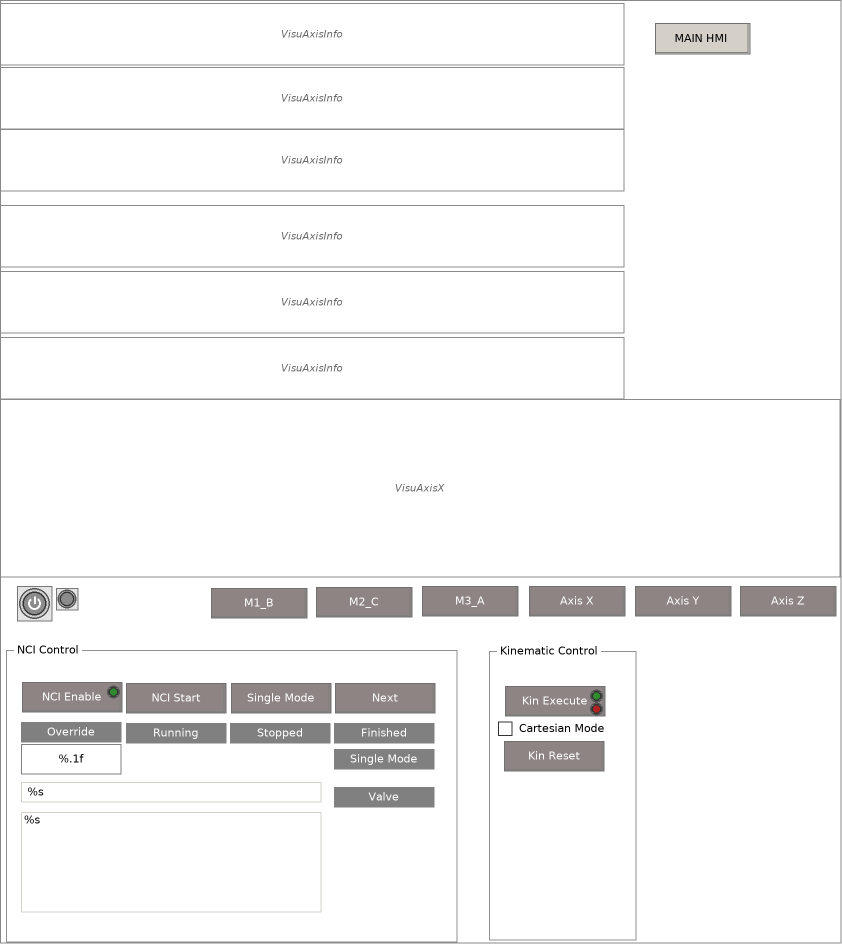
VISUALIZATION Visualization  // 842x944
    Frame (0,205 624x62)
        shows VisuAxisInfo(sAxisName := sAxisXName, stAxisRefVisu := AxisX)
    Frame (0,271 624x62)
        shows VisuAxisInfo(sAxisName := sAxisYName, stAxisRefVisu := AxisY)
    Frame (0,337 624x62)
        shows VisuAxisInfo(sAxisName := sAxisZName, stAxisRefVisu := AxisZ)
    Frame (0,399 840x178)
        shows VisuAxisX()
        shows VisuAxisY()
        shows VisuAxisZ()
        shows VisuAxisM1()
        shows VisuAxisM2()
        shows VisuAxisM3()
    Button (529,586 96x30), "Axis X"
        OnMouseClick: FrameSelectionChange Selection=SelectedFrame=c36eaae5-f889-4027-b551-56d3c927f334, GlobSel=AssignType=Directly, SelType=Locally
    Button (635,586 96x30), "Axis Y"
        OnMouseClick: FrameSelectionChange Selection=SelectedFrame=c36eaae5-f889-4027-b551-56d3c927f334, Selection=1, GlobSel=AssignType=Directly, SelType=Locally
    Button (740,586 96x30), "Axis Z"
        OnMouseClick: FrameSelectionChange Selection=SelectedFrame=c36eaae5-f889-4027-b551-56d3c927f334, Selection=2, GlobSel=AssignType=Directly, SelType=Locally
    GroupBox (6,642 451x300), "NCI Control"
        Button (16,40 100x30), "NCI Enable"
            toggle PRG_NcControl.bNciEnable
        Textfield (15,170 300x100), "%s", text variable: PRG_NcControl.sNciLines
        Button (225,41 100x30), "Single Mode"
            toggle PRG_NcControl.bNciSingleMode
        Rectangle (15,102 100x30), "%.1f", text variable: PRG_NcControl.fNciOverride
            OnMouseClick: write the text variable via VisuDialogs.Numpad
        Rectangle (15,80 100x20), "Override"
        Rectangle (120,81 100x20), "Running", colour toggle: PRG_NcControl.bProgramRunning
        Rectangle (224,81 100x20), "Stopped", colour toggle: PRG_NcControl.bProgramStopped
        Rectangle (328,81 100x20), "Finished", colour toggle: PRG_NcControl.bProgramFinished
        Rectangle (328,145 100x20), "Valve", colour toggle: PRG_MFuncControl.bTestValveOutput
        Button (120,41 100x30), "NCI Start"
            toggle PRG_NcControl.bNciStart
        Button (329,41 100x30), "Next"
            tap PRG_NcControl.bNciNextStep
        Rectangle (328,107 100x20), "Single Mode", colour toggle: PRG_NcControl.bSingleModeActive
        Lamp1 (100,42 15x16), variable: PRG_NcControl.bBuildGroupDone, style: Lamp-Lamp1-Green
    Textfield (21,782 300x20), "%s", text variable: PRG_NcControl.sNciActualLine
    Frame (0,3 624x62)
        shows VisuAxisInfo(sAxisName := sAxisM1_BName, stAxisRefVisu := AxisM1_B)
    Frame (0,67 624x62)
        shows VisuAxisInfo(sAxisName := sAxisM2_CName, stAxisRefVisu := AxisM2_C)
    Frame (0,129 624x62)
        shows VisuAxisInfo(sAxisName := sAxisM3_AName, stAxisRefVisu := AxisM3_A)
    Button (422,586 96x30), "M3_A"
        OnMouseClick: FrameSelectionChange Selection=SelectedFrame=c36eaae5-f889-4027-b551-56d3c927f334, Selection=5, GlobSel=AssignType=Directly, SelType=Locally
    Button (316,587 96x30), "M2_C"
        OnMouseClick: FrameSelectionChange Selection=SelectedFrame=c36eaae5-f889-4027-b551-56d3c927f334, Selection=4, GlobSel=AssignType=Directly, SelType=Locally
    Button (211,588 96x30), "M1_B"
        OnMouseClick: FrameSelectionChange Selection=SelectedFrame=c36eaae5-f889-4027-b551-56d3c927f334, Selection=3, GlobSel=AssignType=Directly, SelType=Locally
    GroupBox (489,643 147x297), "Kinematic Control"
        Button (16,43 100x30), "Kin Execute"
            tap PRG_Kinematic.bExecuteKinConfigGroup
        Checkbox (7,76 119x19), "Cartesian Mode", variable: PRG_Kinematic.bCartesianMode
        Button (15,98 100x30), "Kin Reset"
            tap PRG_Kinematic.bExecuteKinResetGroup
        Lamp1 (100,45 15x16), variable: PRG_Kinematic.fbKinConfigGroup.eKinStatus = KinStatus_Ready, style: Lamp-Lamp1-Green
        Lamp1 (100,58 15x16), variable: PRG_Kinematic.fbKinConfigGroup.bError, invisible if: not PRG_Kinematic.fbKinConfigGroup.bError, style: Lamp-Lamp1-Red
    PowerSwitch (17,586 35x35), variable: GVL_Process.bAllAxesEnable, behaviour: TOGGLE, style: Switch-PowerSwitch-Gray
    PushSwitch (54,588 26x22), variable: GVL_Process.bAllAxesReset, behaviour: TAP, style: Switch-PushSwitch-Gray
    Button (655,23 95x31), "MAIN HMI"
        OnMouseClick: change screen: Visualization_AxesInfo_Manual
END_VISUALIZATION

(* stored: Version 1.1.0.1, ProductVersion 3.1.4022.6
   Visu Visualization: Id {3c523e23-5398-4403-a635-a2cdf8dcb840} *)
